TYPE SC_BUSY_FirstFloor :
(
	enum_member := 0
);
END_TYPE

(* stored: Version 1.1.0.1, ProductVersion 3.1.4024.2
   DUT SC_BUSY_FirstFloor: Id {2e192d48-fe21-4d28-8e90-cef123125fd6} *)
